(* Logix 5000 project; controller TBEN_Lx_8IOL_AOI_V0_2 vendor 1 type 14 code 176 rev 32.11; software revision 32.00; part 16 of 16 *)
(* tags used below, declared in another part *)
   Port : INT;
   Write_Application_Specific_Tag : BOOL;
   Universal_IOLink_Info : Universal_IOLink_Info;
   StartupDone : BOOL;
   Done : DINT;
   Error : DINT;
   Active : DINT;
   Pending : DINT;
   Pending_or_Active : DINT;
   MyTicketNum : DINT[32];
   Read_ONS : DINT;
   ReadRequest : DINT;
   Read : DINT;
   DoneCount : DINT;
   Status : DINT;
   ErrorCount : DINT;
   Prev_Vendor_ID : INT;
   Update_Data : BOOL;
   Write_ONS : DINT;
   WriteRequest : DINT;
(* Universal_Device_Info, continued *)

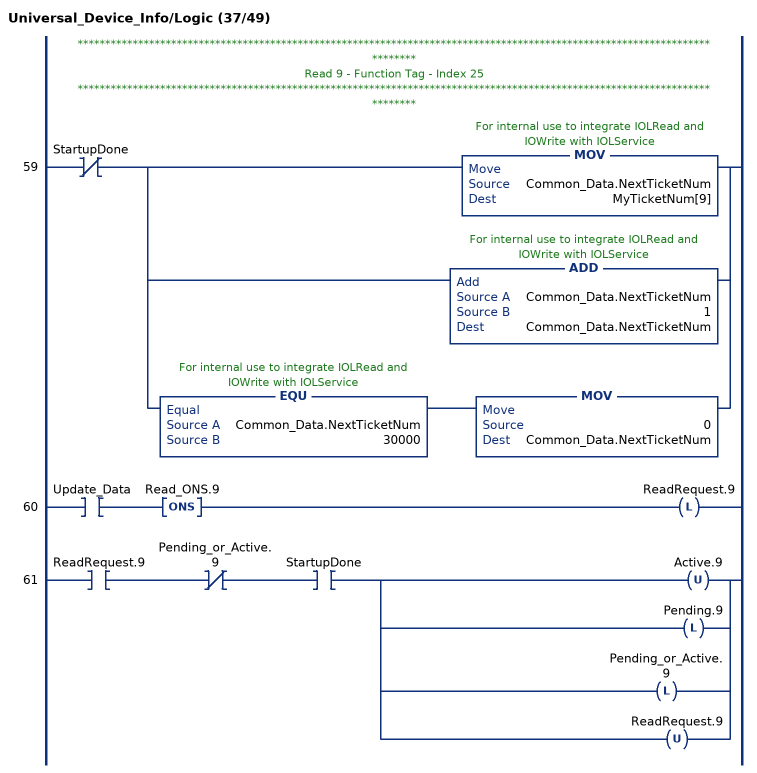
   [picture p85: Universal_Device_Info/Logic rungs 59-61]
   // ***************************************************************************************************************************
   // Read 9 - Function Tag - Index 25
   // ***************************************************************************************************************************
   59: XIO(StartupDone)[MOV(Common_Data.NextTicketNum,MyTicketNum[9]) ,ADD(Common_Data.NextTicketNum,1,Common_Data.NextTicketNum) ,EQU(Common_Data.NextTicketNum,30000) MOV(0,Common_Data.NextTicketNum) ];
   60: XIC(Update_Data)ONS(Read_ONS.9)OTL(ReadRequest.9);
   61: XIC(ReadRequest.9)XIO(Pending_or_Active.9)XIC(StartupDone)[OTU(Active.9) ,OTL(Pending.9) ,OTL(Pending_or_Active.9) ,OTU(ReadRequest.9) ];
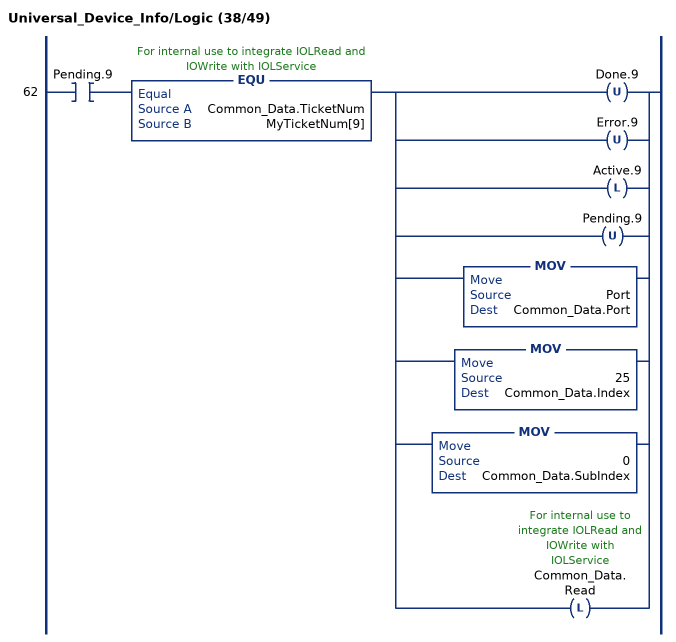
   62: XIC(Pending.9)EQU(Common_Data.TicketNum,MyTicketNum[9])[OTU(Done.9) ,OTU(Error.9) ,OTL(Active.9) ,OTU(Pending.9) ,MOV(Port,Common_Data.Port) ,MOV(25,Common_Data.Index) ,MOV(0,Common_Data.SubIndex) ,OTL(Common_Data.Read) ];
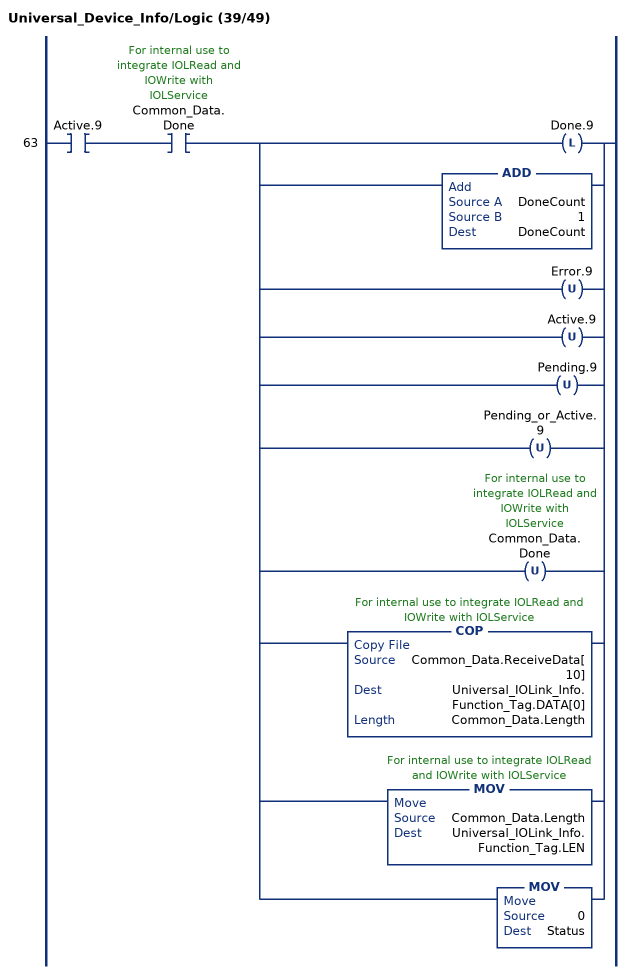
   63: XIC(Active.9)XIC(Common_Data.Done)[OTL(Done.9) ,ADD(DoneCount,1,DoneCount) ,OTU(Error.9) ,OTU(Active.9) ,OTU(Pending.9) ,OTU(Pending_or_Active.9) ,OTU(Common_Data.Done) ,COP(Common_Data.ReceiveData[10],Universal_IOLink_Info.Function_Tag.DATA[0],Common_Data.Length) ,MOV(Common_Data.Length,Universal_IOLink_Info.Function_Tag.LEN) ,MOV(0,Status) ];
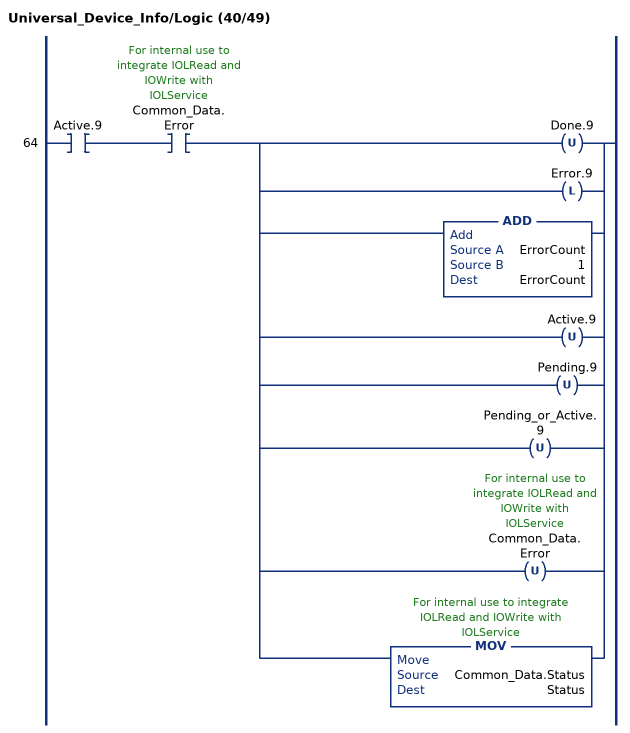
   64: XIC(Active.9)XIC(Common_Data.Error)[OTU(Done.9) ,OTL(Error.9) ,ADD(ErrorCount,1,ErrorCount) ,OTU(Active.9) ,OTU(Pending.9) ,OTU(Pending_or_Active.9) ,OTU(Common_Data.Error) ,MOV(Common_Data.Status,Status) ];
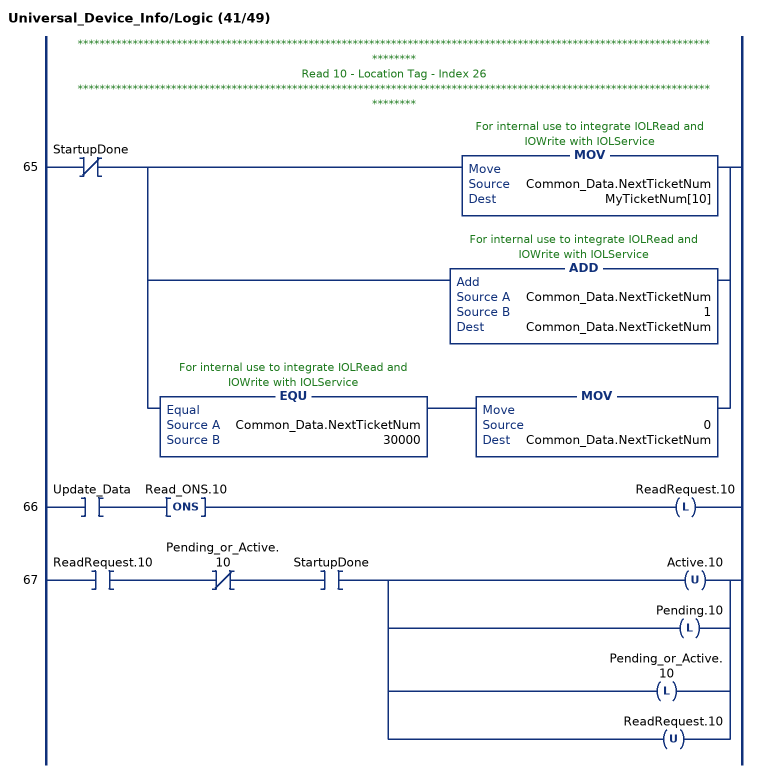
   // ***************************************************************************************************************************
   // Read 10 - Location Tag - Index 26
   // ***************************************************************************************************************************
   65: XIO(StartupDone)[MOV(Common_Data.NextTicketNum,MyTicketNum[10]) ,ADD(Common_Data.NextTicketNum,1,Common_Data.NextTicketNum) ,EQU(Common_Data.NextTicketNum,30000) MOV(0,Common_Data.NextTicketNum) ];
   66: XIC(Update_Data)ONS(Read_ONS.10)OTL(ReadRequest.10);
   67: XIC(ReadRequest.10)XIO(Pending_or_Active.10)XIC(StartupDone)[OTU(Active.10) ,OTL(Pending.10) ,OTL(Pending_or_Active.10) ,OTU(ReadRequest.10) ];
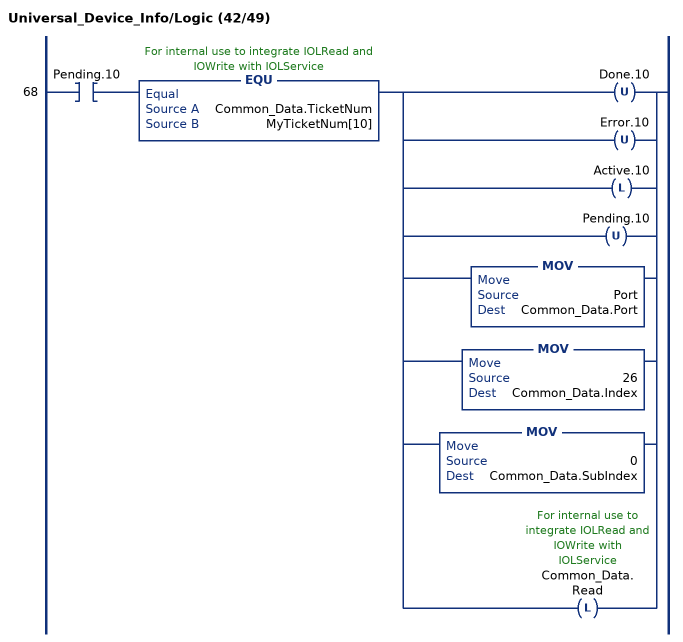
   68: XIC(Pending.10)EQU(Common_Data.TicketNum,MyTicketNum[10])[OTU(Done.10) ,OTU(Error.10) ,OTL(Active.10) ,OTU(Pending.10) ,MOV(Port,Common_Data.Port) ,MOV(26,Common_Data.Index) ,MOV(0,Common_Data.SubIndex) ,OTL(Common_Data.Read) ];
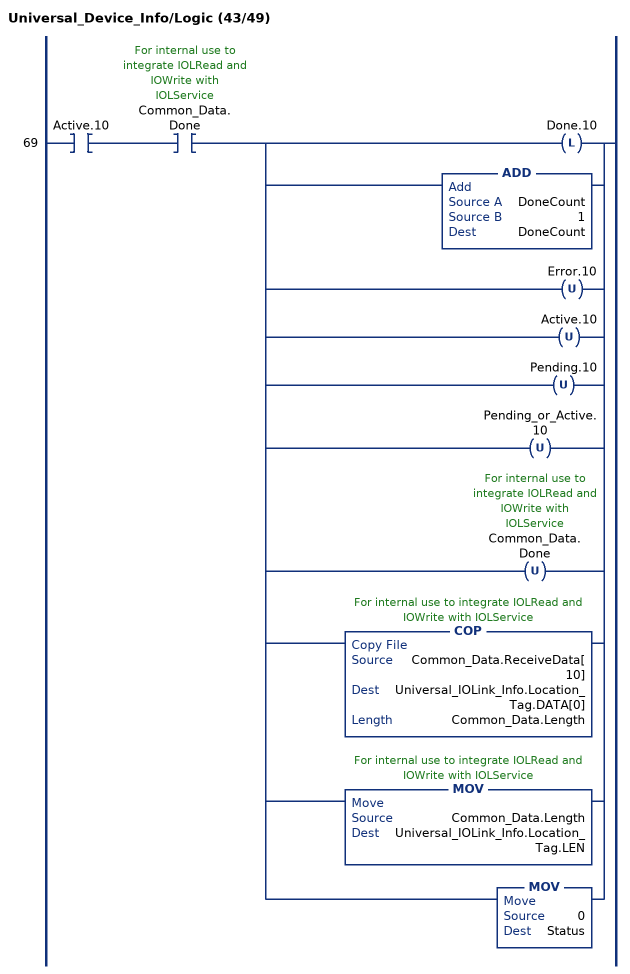
   69: XIC(Active.10)XIC(Common_Data.Done)[OTL(Done.10) ,ADD(DoneCount,1,DoneCount) ,OTU(Error.10) ,OTU(Active.10) ,OTU(Pending.10) ,OTU(Pending_or_Active.10) ,OTU(Common_Data.Done) ,COP(Common_Data.ReceiveData[10],Universal_IOLink_Info.Location_Tag.DATA[0],Common_Data.Length) ,MOV(Common_Data.Length,Universal_IOLink_Info.Location_Tag.LEN) ,MOV(0,Status) ];
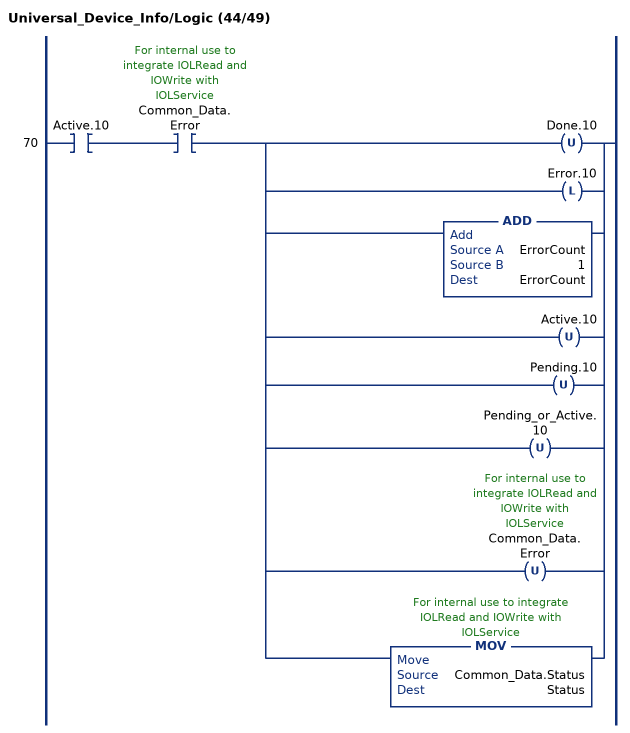
   70: XIC(Active.10)XIC(Common_Data.Error)[OTU(Done.10) ,OTL(Error.10) ,ADD(ErrorCount,1,ErrorCount) ,OTU(Active.10) ,OTU(Pending.10) ,OTU(Pending_or_Active.10) ,OTU(Common_Data.Error) ,MOV(Common_Data.Status,Status) ];
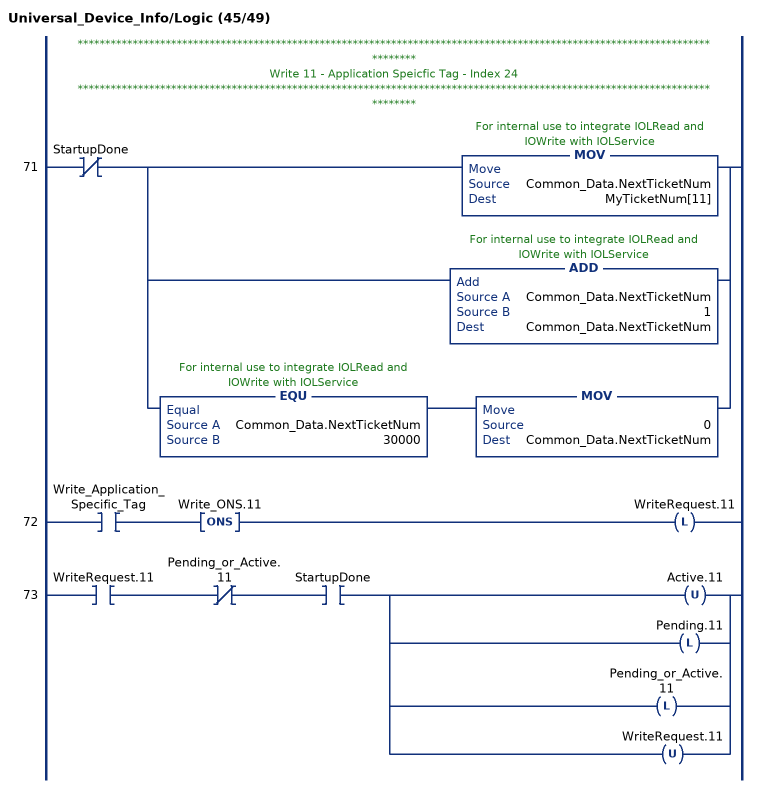
   // ***************************************************************************************************************************
   // Write 11 - Application Speicfic Tag - Index 24
   // ***************************************************************************************************************************
   71: XIO(StartupDone)[MOV(Common_Data.NextTicketNum,MyTicketNum[11]) ,ADD(Common_Data.NextTicketNum,1,Common_Data.NextTicketNum) ,EQU(Common_Data.NextTicketNum,30000) MOV(0,Common_Data.NextTicketNum) ];
   72: XIC(Write_Application_Specific_Tag)ONS(Write_ONS.11)OTL(WriteRequest.11);
   73: XIC(WriteRequest.11)XIO(Pending_or_Active.11)XIC(StartupDone)[OTU(Active.11) ,OTL(Pending.11) ,OTL(Pending_or_Active.11) ,OTU(WriteRequest.11) ];
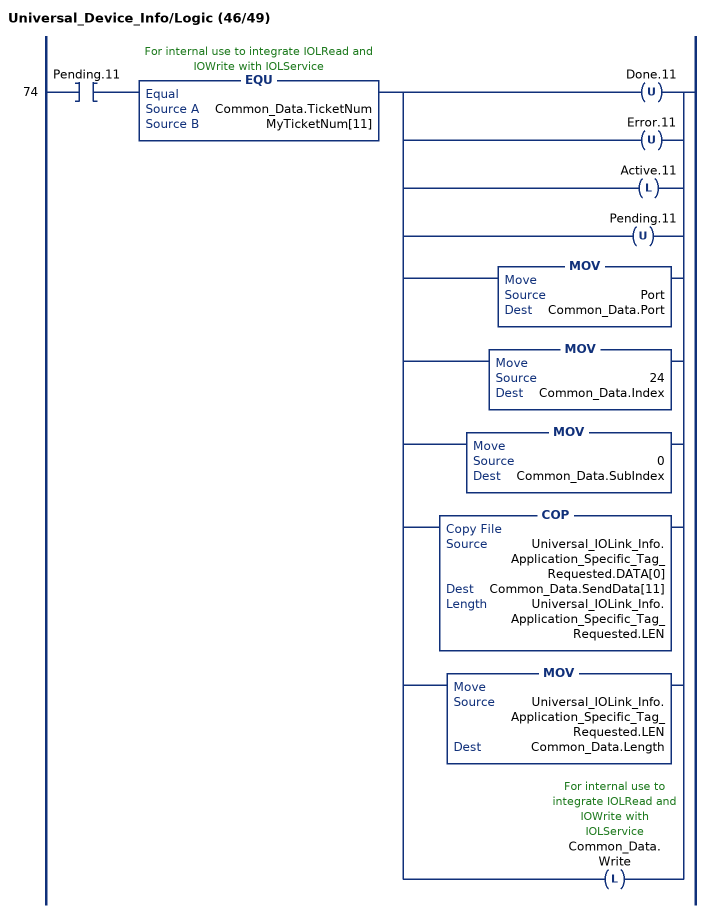
   74: XIC(Pending.11)EQU(Common_Data.TicketNum,MyTicketNum[11])[OTU(Done.11) ,OTU(Error.11) ,OTL(Active.11) ,OTU(Pending.11) ,MOV(Port,Common_Data.Port) ,MOV(24,Common_Data.Index) ,MOV(0,Common_Data.SubIndex) ,COP(Universal_IOLink_Info.Application_Specific_Tag_Requested.DATA[0],Common_Data.SendData[11],Universal_IOLink_Info.Application_Specific_Tag_Requested.LEN) ,MOV(Universal_IOLink_Info.Application_Specific_Tag_Requested.LEN,Common_Data.Length) ,OTL(Common_Data.Write) ];
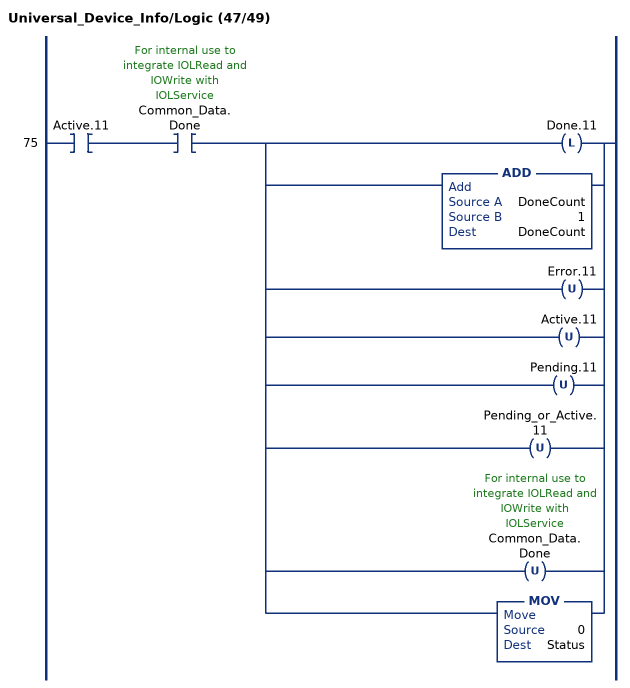
   75: XIC(Active.11)XIC(Common_Data.Done)[OTL(Done.11) ,ADD(DoneCount,1,DoneCount) ,OTU(Error.11) ,OTU(Active.11) ,OTU(Pending.11) ,OTU(Pending_or_Active.11) ,OTU(Common_Data.Done) ,MOV(0,Status) ];
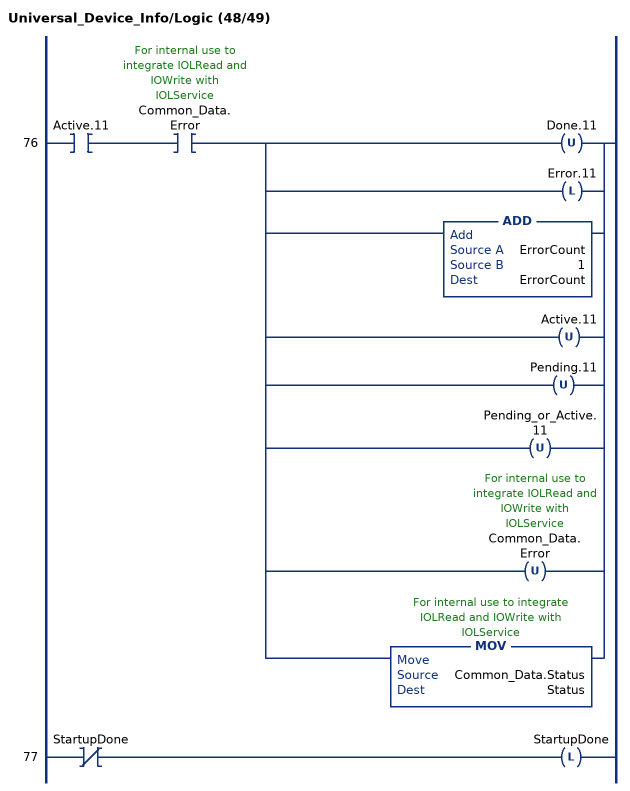
   76: XIC(Active.11)XIC(Common_Data.Error)[OTU(Done.11) ,OTL(Error.11) ,ADD(ErrorCount,1,ErrorCount) ,OTU(Active.11) ,OTU(Pending.11) ,OTU(Pending_or_Active.11) ,OTU(Common_Data.Error) ,MOV(Common_Data.Status,Status) ];
   77: XIO(StartupDone)OTL(StartupDone);
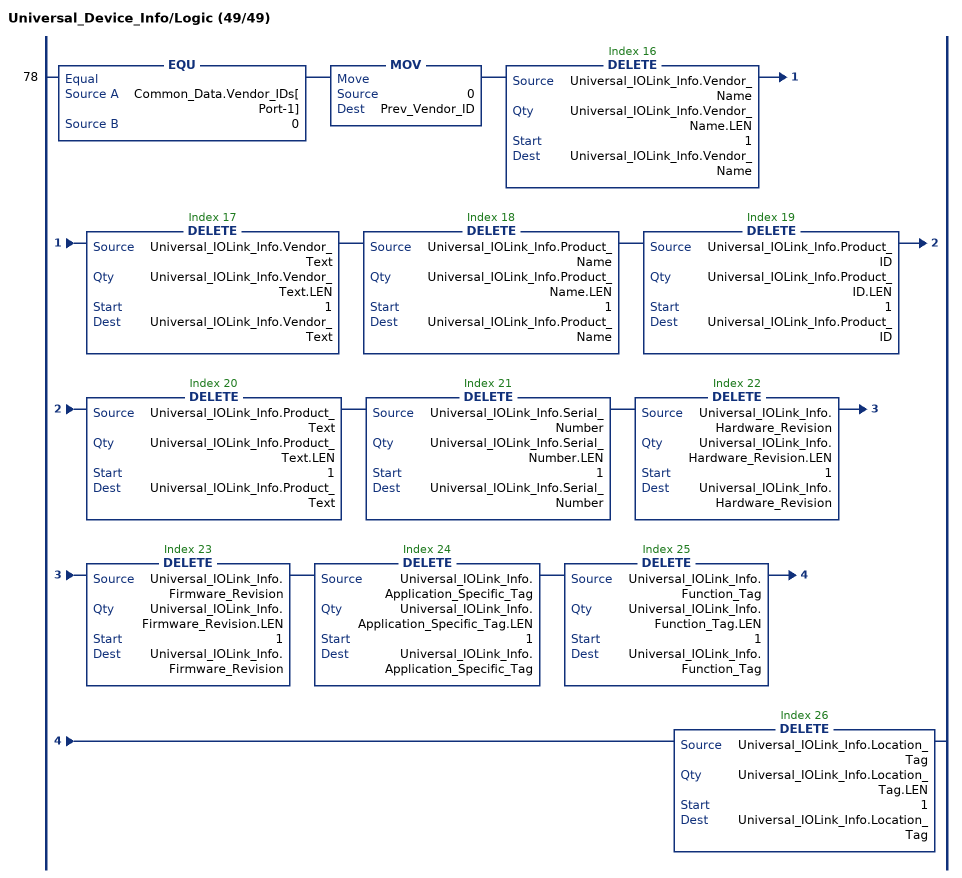
   78: EQU(Common_Data.Vendor_IDs[Port-1],0)MOV(0,Prev_Vendor_ID)DELETE(Universal_IOLink_Info.Vendor_Name,Universal_IOLink_Info.Vendor_Name.LEN,1,Universal_IOLink_Info.Vendor_Name)DELETE(Universal_IOLink_Info.Vendor_Text,Universal_IOLink_Info.Vendor_Text.LEN,1,Universal_IOLink_Info.Vendor_Text)DELETE(Universal_IOLink_Info.Product_Name,Universal_IOLink_Info.Product_Name.LEN,1,Universal_IOLink_Info.Product_Name)DELETE(Universal_IOLink_Info.Product_ID,Universal_IOLink_Info.Product_ID.LEN,1,Universal_IOLink_Info.Product_ID)DELETE(Universal_IOLink_Info.Product_Text,Universal_IOLink_Info.Product_Text.LEN,1,Universal_IOLink_Info.Product_Text)DELETE(Universal_IOLink_Info.Serial_Number,Universal_IOLink_Info.Serial_Number.LEN,1,Universal_IOLink_Info.Serial_Number)DELETE(Universal_IOLink_Info.Hardware_Revision,Universal_IOLink_Info.Hardware_Revision.LEN,1,Universal_IOLink_Info.Hardware_Revision)DELETE(Universal_IOLink_Info.Firmware_Revision,Universal_IOLink_Info.Firmware_Revision.LEN,1,Universal_IOLink_Info.Firmware_Revision)DELETE(Universal_IOLink_Info.Application_Specific_Tag,Universal_IOLink_Info.Application_Specific_Tag.LEN,1,Universal_IOLink_Info.Application_Specific_Tag)DELETE(Universal_IOLink_Info.Function_Tag,Universal_IOLink_Info.Function_Tag.LEN,1,Universal_IOLink_Info.Function_Tag)DELETE(Universal_IOLink_Info.Location_Tag,Universal_IOLink_Info.Location_Tag.LEN,1,Universal_IOLink_Info.Location_Tag);
END_ROUTINE

ROUTINE Prescan   (* ladder *)
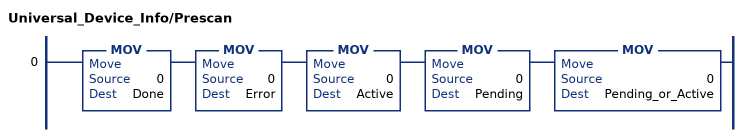
   0: MOV(0,Done)MOV(0,Error)MOV(0,Active)MOV(0,Pending)MOV(0,Pending_or_Active);
END_ROUTINE
END_ADD_ON_INSTRUCTION

VAR_GLOBAL   (* controller tags *)
   Common_Data : Turck_IOLink_Common_Data := (Port := 128, Index := -1, SubIndex := 68, Length := 224, NextTicketNum := 1, ReceiveData[206] := 1, ReceiveData[207] := 61, ReceiveData[209] := 30, ReceiveData[210] := 51, ReceiveData[211] := 3, ReceiveData[214] := 48, ReceiveData[215] := 48, ReceiveData[216] := 48, ReceiveData[217] := 49, ReceiveData[218] := 48, ReceiveData[219] := 55, ReceiveData[220] := 54, ReceiveData[221] := 54, ReceiveData[222] := 53, ReceiveData[223] := 56, ReceiveData[224] := 45, ReceiveData[225] := 48, ReceiveData[226] := 48, ReceiveData[227] := 48, ReceiveData[228] := 50, ReceiveData[229] := 48, ReceiveData[230] := 17, ReceiveData[231] := 16, ReceiveData[232] := 16, ReceiveData[233] := 32, ReceiveData[234] := 45, ReceiveData[235] := 48, ReceiveData[236] := 48, ReceiveData[237] := 48, ReceiveData[238] := 50, ReceiveData[239] := 48, ReceiveData[240] := 17, ReceiveData[241] := 16, ReceiveData[242] := 16, ReceiveData[243] := 32, SendData[0] := -1, SendData[1] := -1, SendData[2] := 68, Vendor_IDs[7] := 317, Device_IDs[7] := 1979139, Process_Input_Data[7].Data[0] := 32);
   IOL_READ_MSG : MESSAGE;
        MessageParameters(ServiceCode := 16#004b, LocalElement := Common_Data.SendData, DestinationTag := Common_Data.ReceiveData, ...)
   IOL_WRITE_MSG : MESSAGE;
        MessageParameters(ServiceCode := 16#004c, LocalElement := Common_Data.SendData, DestinationTag := Common_Data.ReceiveData, ...)
   TBEN_8IOL_101 : TBEN_Lx_8IOL_AOI := (IOLDevice_PORT8 := 1);
   TBEN_8IOL_101_Config_Tags_IN : Generic_160_SINT := (DATA[14] := 1, DATA[15] := 1, DATA[16] := 1, DATA[17] := 1, DATA[25] := 3, DATA[41] := 3, DATA[57] := 3, DATA[73] := 3, DATA[89] := 3, DATA[105] := 3, DATA[121] := 3, DATA[137] := 3);
   TBEN_8IOL_101_Config_Tags_OUT : Generic_160_SINT := (DATA[14] := 1, DATA[15] := 1, DATA[16] := 1, DATA[17] := 1, DATA[25] := 3, DATA[41] := 3, DATA[57] := 3, DATA[73] := 3, DATA[89] := 3, DATA[105] := 3, DATA[121] := 3, DATA[137] := 3);
   TBEN_8IOL_101_Process_Data_In : Generic_173_Words := (Data[2] := 1, Data[3] := 16384);
   TBEN_8IOL_101_Process_Data_Out : Generic_131_Words;
   TBIL : Universal_Device_Info := (Port := 1);
   TBIL_Info : Universal_IOLink_Info;
   TEST : BOOL;
END_VAR

PROGRAM MainProgram   (* main routine MainRoutine *)
VAR
   TBEN_8IOL_100_Process_Data_In : Generic_173_Words := (Data[0] := 1, Data[133] := 4, Data[134] := 4, Data[135] := 4, Data[136] := 4, Data[137] := 4, Data[138] := 4, Data[139] := 4, Data[140] := 4);
   TBEN_8IOL_100_Process_Data_Out : Generic_131_Words;
END_VAR

ROUTINE MainRoutine   (* ladder *)
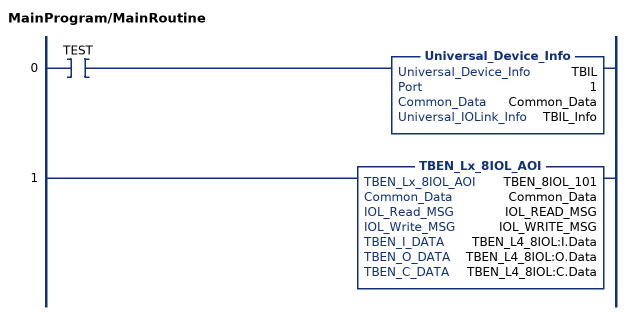
   0: XIC(TEST)Universal_Device_Info(TBIL,1,Common_Data,TBIL_Info);
   1: TBEN_Lx_8IOL_AOI(TBEN_8IOL_101,Common_Data,IOL_READ_MSG,IOL_WRITE_MSG,TBEN_L4_8IOL:I.Data,TBEN_L4_8IOL:O.Data,TBEN_L4_8IOL:C.Data);
END_ROUTINE
END_PROGRAM

PROGRAM SafetyProgram   (* main routine MainRoutine, safety *)

ROUTINE MainRoutine   (* ladder *)
END_ROUTINE
END_PROGRAM
